FUNCTION_BLOCK iterator
VAR_INPUT
	increment	:	DINT;
END_VAR
VAR_OUTPUT
	out	:	DINT;
END_VAR
VAR
	value	:	DINT	:=0;
	lim	:	DINT :=1000;
END_VAR

IF value < lim THEN
	value := value + increment;
ELSE
	value:= 0;	
END_IF
out := value;

END_FUNCTION_BLOCK

(* stored: Version 1.1.0.1, ProductVersion 3.1.4020.12
   POU iterator: Id {f811f75d-3bc1-47ae-8e78-e15fbc0722ce}, SpecialFunc None *)
